INTERFACE iMoverList

METHOD ActivateAllTrack : iMoverList
VAR_INPUT
	Track	: REFERENCE TO Track;
END_VAR
END_METHOD

METHOD GetMoverByLocation : REFERENCE to Mover
VAR_INPUT
    Index     : USINT;                // 0 is find the first closest mover, 1 is find the second closest mover, 2 is find the third, etc. etc. etc.
    Position  : LREAL;                // Fixed track position from which to search for movers by proximity
    Direction : Tc2_MC2.MC_Direction; // Positive = find the most positive mover whose position is less than the Input. Negative = find the most negative mover whose position is greater than the input
END_VAR
END_METHOD

PROPERTY IsAllTrackReady : BOOL
GET
END_GET
END_PROPERTY

METHOD MoveAllToPosition : iMoverList
VAR_INPUT

    DestinationPosition : LREAL; // position on track for all shuttles to move towards	

END_VAR
END_METHOD

METHOD MoveAllToStation : iMoverList
VAR_INPUT

    DestinationStation : REFERENCE TO Station;

END_VAR
END_METHOD

METHOD MoveAllVelocity : iMoverList
VAR_INPUT

    Velocity : LREAL;

END_VAR
END_METHOD

METHOD SetAllAcceleration : iMoverList
VAR_INPUT

    Acceleration : LREAL;

END_VAR
END_METHOD

METHOD SetAllDeceleration : iMoverList
VAR_INPUT

    Deceleration : LREAL;

END_VAR
END_METHOD

METHOD SetAllDirection : iMoverList
VAR_INPUT

    Direction : Tc3_Mc3Definitions.MC_DIRECTION;

END_VAR
END_METHOD

METHOD SetAllJerk : iMoverList
VAR_INPUT

    Jerk : LREAL;

END_VAR
END_METHOD

METHOD SetAllVelocity : iMoverList
VAR_INPUT

    Velocity : LREAL;

END_VAR
END_METHOD

{attribute 'monitoring' := 'call'}
PROPERTY TrackedMoverCount : USINT
GET
END_GET
END_PROPERTY

PROPERTY TrackedMovers : ARRAY[0..GVL.NUM_MOVERS - 1] OF POINTER TO Mover
GET
END_GET
END_PROPERTY

METHOD UnregisterAll : BOOL
VAR_INPUT
END_VAR
END_METHOD

END_INTERFACE

(* stored: Version 1.1.0.1, ProductVersion 3.1.4024.12
   Itf iMoverList: Id {9cc4a2ad-2506-4bdd-acf3-bfbfde25ab77}
   Method ActivateAllTrack: Id {214d853b-c1b8-0faa-14bf-a2670bf33012}
   Method GetMoverByLocation: Id {08ab6dd2-55e6-476a-991b-26d3f0ccc58d}
   Property IsAllTrackReady: Id {a3e4944a-7607-0f5a-10b2-64b1616a1317}
   Get Get: Id {c87cec46-e2a4-0a12-2b5e-a6b05f1caa93}
   Method MoveAllToPosition: Id {745a52d9-fa71-49ff-868a-52a3293e2e2d}
   Method MoveAllToStation: Id {371362e2-fc11-40b6-a0e6-d17b876d5e78}
   Method MoveAllVelocity: Id {be6cc2f7-a0ce-45ef-a956-f19486620100}
   Method SetAllAcceleration: Id {455895b5-97e6-495e-9cb5-6646f55e97b6}
   Method SetAllDeceleration: Id {d14e387e-79be-456d-9c0b-e3f03ddf19f2}
   Method SetAllDirection: Id {4bfb0de3-28b7-4b24-a865-2cf8e65fcd48}
   Method SetAllJerk: Id {a91832af-959e-462a-a423-5a2f3601faa8}
   Method SetAllVelocity: Id {2027ef8a-c9a4-4e95-be1e-4ccdc273c80d}
   Property TrackedMoverCount: Id {368f6c76-4224-03b5-39ed-4f46132302d9}
   Get Get: Id {a4e1bb20-cd42-038c-1a1e-a8f5b0110892}
   Property TrackedMovers: Id {c1d0d30a-4686-4f53-a96b-53d64c99ec16}
   Get Get: Id {d3d3bfad-1918-438f-8ad5-aa73cc840431}
   Method UnregisterAll: Id {77dd6571-5452-49cc-817d-10e46daccff7} *)
